Staubli VAL3: RefreshList.pgx

program RefreshList()
  local num l_ni
begin
  //
  if bListRefresh
    resize(sList,1,20)
    for l_ni=0 to 19
      sList[l_ni]="Frame"+toString("",l_ni+1)
    endFor
  endIf

end
